{attribute 'reflection'}
FUNCTION_BLOCK ABSTRACT T_EventBase IMPLEMENTS I_Event
VAR
    EventHandlers : T_ListOfEventHandlers(Capacity := 5);
    
    {attribute 'instance-path'} {attribute 'no_init'}
    EventName : T_MaxString; // Automatically initialised with the full name of the instance   
    
    EventArgs : T_Stream(StreamLength := 8);
    
    Message_EventHandlerNotImplemented : FB_TcMessage;
END_VAR

METHOD AddEventHandler : I_Event
VAR_INPUT
    Handler : I_EventHandlerBase;
END_VAR
IF IsHandlerSupported(Handler) THEN
    EventHandlers.AddHandler(Handler);
//ELSE
//    IF Message_EventHandlerNotImplemented.nEventId = 0 THEN
//        Message_EventHandlerNotImplemented.CreateEx(
//            stEventEntry := TC_EVENTS.tcl_BaseClassEvents.EventHandlerNotImplemented,
//            ipSourceInfo := 0);
//    END_IF
//    Message_EventHandlerNotImplemented.Send(0);

END_IF
AddEventHandler := THIS^;
END_METHOD

PROPERTY PUBLIC Args : I_StreamWriter
GET
Args := EventArgs;
END_GET
END_PROPERTY

METHOD ABSTRACT CallHandler
VAR_INPUT
    HandlerBase : I_EventHandlerBase;
    EventArgs : I_StreamReader;
END_VAR
END_METHOD

METHOD ClearEventHandlers : I_Event
EventHandlers.Clear();
ClearEventHandlers := THIS^;
END_METHOD

METHOD ABSTRACT IsHandlerSupported : BOOL
VAR_INPUT
    HandlerBase : I_EventHandlerBase;
END_VAR
END_METHOD

METHOD Raise
VAR
    HandlerBase : I_EventHandlerBase;
    i : UDINT;
END_VAR
IF EventHandlers.Count > 0 THEN
    FOR i := 0 TO EventHandlers.Count - 1 DO
        HandlerBase := EventHandlers.GetHandler(i);
        IF HandlerBase <> 0 THEN
            EventArgs.Seek(0); // to ensure that each handler reads args from start of the stream
            CallHandler(HandlerBase,EventArgs);
        END_IF
    END_FOR
END_IF
EventArgs.Clear(); // to leave event args empty for next time event is raised
END_METHOD

END_FUNCTION_BLOCK

(* stored: Version 1.1.0.1, ProductVersion 3.1.4024.4
   POU T_EventBase: Id {720ebf79-c150-0ee1-0a2c-8a2b014bb121}, SpecialFunc None
   Method AddEventHandler: Id {fac94ceb-09e8-0c42-3422-f61b79869355}
   Property Args: Id {a18ec44b-b2bb-0d6e-00e1-3cc9afdf8f65}
   Get Get: Id {131c9f6c-d685-0dc6-0c2d-8edfc67e855a}
   Method CallHandler: Id {d21491e4-062a-0729-1d4a-7c6d64c8e4e5}
   Method ClearEventHandlers: Id {4cb8b6ff-767b-0ea6-0e34-89f3978cdefb}
   Method IsHandlerSupported: Id {539bb4e2-623c-0ec0-3e41-d67563c031d7}
   Method Raise: Id {e0f1ad27-77a6-08d5-08c8-71ccdfdf6f90} *)
